PROGRAM simIniciaProg
VAR
	bSimIniciaProg: BOOL:= FALSE;
	posicaoAtual: STRING;
	envialog: STRING;
	bGravarConfigPosicao_Reator: BOOL;
END_VAR


gvl_p.arrStatusEstufas[gvl.actEst].start := TRUE;

bGravarConfigPosicao_Reator:= TRUE;

END_PROGRAM

(* stored: Version 1.1.0.1, ProductVersion 3.1.4024.12
   POU simIniciaProg: Id {662f6976-2ee6-4828-b8d3-9fbd7250e3cb}, SpecialFunc None *)
